FUNCTION_BLOCK FB_Component_DualValve IMPLEMENTS I_Component
VAR_INPUT
	sName			: STRING[50];
	tTimeout		: TIME := T#0S;
END_VAR

VAR_IN_OUT
	bOutputA		: BOOL;
	bOutputB		: BOOL;
END_VAR

VAR_OUTPUT
	bEnabled     	: BOOL;
	eState			: E_State;
	sStatusText 	: STRING[100];
END_VAR

VAR
	bStartTimeout	: BOOL;
	tTimeoutTimer	: TON;
	bLastOutputA	: BOOL;
	bLastOutputB	: BOOL;
	eLastState		: E_State;
END_VAR

VAR CONSTANT
	DISABLED		: E_State := E_State.DISABLED;
	READY			: E_State := E_State.READY;
	BUSY			: E_State := E_State.BUSY;
	DONE			: E_State := E_State.DONE;
	HALTED			: E_State := E_State.HALTED;
	TIMEOUT			: E_State := E_State.TIMEOUT;
END_VAR

tTimeoutTimer(PT := tTimeout);

CASE eState OF
	DISABLED: 	sStatusText := 'piston disabled';
	READY: 		sStatusText := 'piston ready to operate';
	BUSY: 		sStatusText := '';
	
	TIMEOUT:	sStatusText := 'piston in timeout';
				tTimeoutTimer(IN := TRUE);
				
				IF tTimeoutTimer.Q THEN
					eState := E_State.DONE;
				END_IF
				
	DONE:		sStatusText := 'piston done';
				tTimeoutTimer(IN := FALSE);
				M_Resume();
	HALTED:		sStatusText := 'piston halted';
END_CASE

METHOD M_Disable : BOOL
VAR_INPUT
END_VAR
IF eState = DONE OR eState = READY THEN
	bEnabled	:= FALSE;
	eState		:= DISABLED;
END_IF
END_METHOD

METHOD M_Enable : BOOL
VAR_INPUT
END_VAR
IF eState = DISABLED THEN
	bEnabled	:= TRUE;
	eState 		:= READY;
END_IF
END_METHOD

METHOD M_Extend : BOOL
VAR_INPUT
END_VAR
IF eState = READY OR eState = BUSY THEN
	bOutputA	:= TRUE;
	bOutputB	:= FALSE;
END_IF
END_METHOD

METHOD M_Halt : BOOL
VAR_INPUT
END_VAR
bOutputA		:= FALSE;
bOutputB		:= FALSE;
bLastOutputA	:= bOutputA;
bLastOutputB	:= bOutputB;
eLastState 		:= eState;
eState 			:= HALTED;
END_METHOD

METHOD M_Hold : BOOL
VAR_INPUT
END_VAR
IF eState = READY OR eState = BUSY THEN
	bOutputA	:= FALSE;
	bOutputB	:= FALSE;
	eState 		:= TIMEOUT;
END_IF
END_METHOD

METHOD M_Reset : BOOL
VAR_INPUT
END_VAR
// has no use here
END_METHOD

METHOD M_Resume : BOOL
VAR_INPUT
END_VAR
CASE eState OF
	HALTED	: 	bOutputA	:= bLastOutputA;
				bOutputB	:= bLastOutputB;
				eState 		:= eLastState;
				
	DONE	: 	eState 		:= READY;
END_CASE
END_METHOD

METHOD M_Retract : BOOL
VAR_INPUT
END_VAR
IF eState = READY OR eState = BUSY THEN
	bOutputA	:= FALSE;
	bOutputB	:= TRUE;
END_IF
END_METHOD

METHOD M_Stop : BOOL
VAR_INPUT
END_VAR
IF eState <> BUSY OR eState <> HALTED OR eState <> TIMEOUT THEN
	bOutputA	:= FALSE;
	bOutputB	:= FALSE;
	eState 		:= DONE;
END_IF
END_METHOD

END_FUNCTION_BLOCK

(* stored: Version 1.1.0.1, ProductVersion 3.1.4024.15
   POU FB_Component_DualValve: Id {04d6caaa-12ea-4ca7-b40e-e6e2c47167ec}, SpecialFunc None
   Method M_Disable: Id {857ba533-460d-49df-a434-29ec9866f2c4}
   Method M_Enable: Id {5572c232-6e47-4666-97bc-7f38e6278500}
   Method M_Extend: Id {652675af-aaae-439e-b0a9-8329efd7407d}
   Method M_Halt: Id {1ef68817-4258-41df-bb9a-e1887637bbb5}
   Method M_Hold: Id {e1e0c979-5fbf-42d6-a4c4-75167087b8ec}
   Method M_Reset: Id {1ce6f44c-2ddc-4921-b544-bc588c6a8184}
   Method M_Resume: Id {9c7a6fbd-0999-4d44-a452-a166548a9afa}
   Method M_Retract: Id {9551191d-fe4d-4d72-b2a9-7e17fb7d2b9c}
   Method M_Stop: Id {49386caf-422f-4ba8-a140-e94b68e1642d} *)
